SUBAPPLICATION GesamtzaehlerVergleich (* Subapplication Type *)
  (* Standard: 61499-2 *)
  (* Version 1.0, 2023-02-18, Franz *)
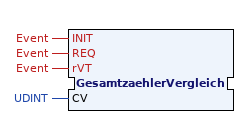
  EVENT_INPUT
    INIT; (* Initialization Request *)
    REQ; (* Normal Execution Request *)
    rVT; (* refresh VT *)
  END_EVENT
  VAR_INPUT
    CV : UDINT; (* Counter Value *)
  END_VAR
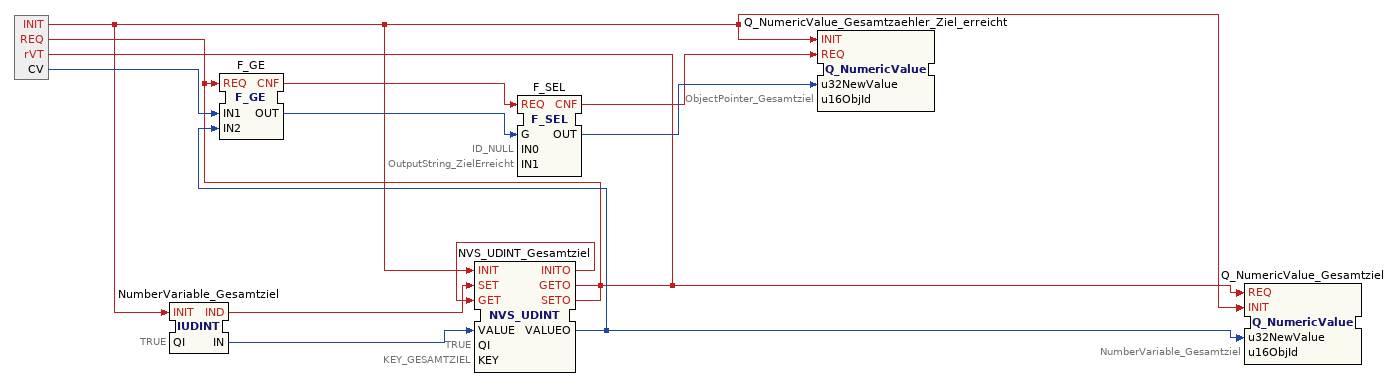
  FBS
    Q_NumericValue_Gesamtzaehler_Ziel_erreicht : Q_NumericValue(u16ObjId := ObjectPointer_Gesamtziel);
    F_GE : F_GE;
    NVS_UDINT_Gesamtziel : NVS_UDINT(QI := TRUE, KEY := KEY_GESAMTZIEL);
    NumberVariable_Gesamtziel : IUDINT(QI := TRUE);
    Q_NumericValue_Gesamtziel : Q_NumericValue(u16ObjId := NumberVariable_Gesamtziel);
    F_SEL : F_SEL(IN0 := ID_NULL, IN1 := OutputString_ZielErreicht);
  END_FBS
  EVENT_CONNECTIONS
    INIT TO Q_NumericValue_Gesamtzaehler_Ziel_erreicht.INIT;
    REQ TO F_GE.REQ;
    INIT TO NumberVariable_Gesamtziel.INIT;
    INIT TO NVS_UDINT_Gesamtziel.INIT;
    NumberVariable_Gesamtziel.IND TO NVS_UDINT_Gesamtziel.SET;
    NVS_UDINT_Gesamtziel.INITO TO NVS_UDINT_Gesamtziel.GET;
    NVS_UDINT_Gesamtziel.GETO TO Q_NumericValue_Gesamtziel.REQ;
    INIT TO Q_NumericValue_Gesamtziel.INIT;
    NVS_UDINT_Gesamtziel.GETO TO F_GE.REQ;
    NVS_UDINT_Gesamtziel.SETO TO F_GE.REQ;
    rVT TO Q_NumericValue_Gesamtziel.REQ;
    F_GE.CNF TO F_SEL.REQ;
    F_SEL.CNF TO Q_NumericValue_Gesamtzaehler_Ziel_erreicht.REQ;
  END_CONNECTIONS
  DATA_CONNECTIONS
    CV TO F_GE.IN1;
    NumberVariable_Gesamtziel.IN TO NVS_UDINT_Gesamtziel.VALUE;
    NVS_UDINT_Gesamtziel.VALUEO TO Q_NumericValue_Gesamtziel.u32NewValue;
    NVS_UDINT_Gesamtziel.VALUEO TO F_GE.IN2;
    F_GE.OUT TO F_SEL.G;
    F_SEL.OUT TO Q_NumericValue_Gesamtzaehler_Ziel_erreicht.u32NewValue;
  END_CONNECTIONS
END_SUBAPPLICATION
